FUNCTION_BLOCK ThreeConveyor (* Composite Function Block Type *)
  (* Standard: 61499-2 *)
  (* Version 0.2, 2003-12-05, JHC, Rockwell Automation, Renamed from NEWCOMPFB. *)
  (* Version 0.1, 2002-01-08, JHC, Rockwell Automation, Added DLY FB as example. *)
  (* Version 0.0, 2000-05-27, JHC, Rockwell Automation *)
  (* Compiler header: package fb.rt.cs725; *)
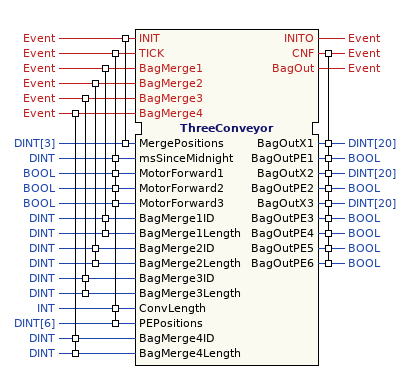
  EVENT_INPUT
    INIT WITH MergePositions; (* Initialization Request *)
    TICK WITH msSinceMidnight, MotorForward1, MotorForward2, MotorForward3, ConvLength, PEPositions; (* Normal Execution Request *)
    BagMerge1 WITH BagMerge1ID, BagMerge1Length;
    BagMerge2 WITH BagMerge2ID, BagMerge2Length;
    BagMerge3 WITH BagMerge3ID, BagMerge3Length;
    BagMerge4 WITH BagMerge4ID, BagMerge4Length;
  END_EVENT
  EVENT_OUTPUT
    INITO; (* Initialization Confirm *)
    CNF WITH BagOutX1, BagOutPE1, BagOutX2, BagOutPE2, BagOutX3, BagOutPE3, BagOutPE4, BagOutPE5, BagOutPE6; (* Execution Confirmation *)
    BagOut;
  END_EVENT
  VAR_INPUT
    MergePositions : ARRAY [0..2] OF DINT;
    msSinceMidnight : DINT;
    MotorForward1 : BOOL;
    MotorForward2 : BOOL;
    MotorForward3 : BOOL;
    BagMerge1ID : DINT;
    BagMerge1Length : DINT;
    BagMerge2ID : DINT;
    BagMerge2Length : DINT;
    BagMerge3ID : DINT;
    BagMerge3Length : DINT;
    ConvLength : INT;
    PEPositions : ARRAY [0..5] OF DINT;
    BagMerge4ID : DINT;
    BagMerge4Length : DINT;
  END_VAR
  VAR_OUTPUT
    BagOutX1 : ARRAY [0..19] OF DINT;
    BagOutPE1 : BOOL;
    BagOutX2 : ARRAY [0..19] OF DINT;
    BagOutPE2 : BOOL;
    BagOutX3 : ARRAY [0..19] OF DINT;
    BagOutPE3 : BOOL;
    BagOutPE4 : BOOL;
    BagOutPE5 : BOOL;
    BagOutPE6 : BOOL;
  END_VAR
  FBS
    C1 : Conveyor_Model_WithNetwork;
    C2 : Conveyor_Model_WithNetwork;
    C3 : Conveyor_Model_WithNetwork;
  END_FBS
  EVENT_CONNECTIONS
    INIT TO C1.INIT;
    TICK TO C1.TICK;
    BagMerge1 TO C1.BagMerge1;
    BagMerge3 TO C1.BagMerge2;
    C1.BagOut TO C2.BagIn;
    C1.CNF TO C2.TICK;
    C1.INITO TO C2.INIT;
    C2.INITO TO C3.INIT;
    C2.CNF TO C3.TICK;
    C2.BagOut TO C3.BagIn;
    C3.INITO TO INITO;
    C3.CNF TO CNF;
    BagMerge2 TO C2.BagMerge1;
    BagMerge4 TO C3.BagMerge1;
  END_CONNECTIONS
  DATA_CONNECTIONS
    ConvLength TO C1.ConvLength;
    PEPositions TO C1.PEPositions;
    MergePositions TO C1.MergePositions;
    msSinceMidnight TO C1.msSinceMidnight;
    MotorForward1 TO C1.MotorForward;
    BagMerge1ID TO C1.BagMerge1ID;
    BagMerge1Length TO C1.BagMerge1Length;
    BagMerge3ID TO C1.BagMerge2ID;
    BagMerge3Length TO C1.BagMerge2Length;
    ConvLength TO C2.ConvLength;
    PEPositions TO C2.PEPositions;
    MergePositions TO C2.MergePositions;
    C1.BagOutID TO C2.BagInID;
    C1.BagOutLength TO C2.BagInLength;
    C2.BagOutID TO C3.BagInID;
    C2.BagOutLength TO C3.BagInLength;
    msSinceMidnight TO C2.msSinceMidnight;
    MotorForward2 TO C2.MotorForward;
    BagMerge2ID TO C2.BagMerge1ID;
    BagMerge2Length TO C2.BagMerge1Length;
    ConvLength TO C3.ConvLength;
    PEPositions TO C3.PEPositions;
    MergePositions TO C3.MergePositions;
    msSinceMidnight TO C3.msSinceMidnight;
    MotorForward3 TO C3.MotorForward;
    C1.BagOutX TO BagOutX1;
    C2.BagOutX TO BagOutX2;
    C3.BagOutX TO BagOutX3;
    C1.BagOutPE TO BagOutPE4;
    C2.BagOutPE TO BagOutPE5;
    C1.BagOutPE2 TO BagOutPE1;
    C2.BagOutPE2 TO BagOutPE2;
    C3.BagOutPE2 TO BagOutPE3;
    BagMerge4ID TO C3.BagMerge1ID;
    BagMerge4Length TO C3.BagMerge1Length;
    C3.BagOutPE TO BagOutPE6;
  END_CONNECTIONS
END_FUNCTION_BLOCK
